Omron CX-Programmer project NuevoProyecto (CX-Programmer ?)

# PLC NuevoPLC1: CPM1(CPM1A) CPU30

## Program NuevoPrograma1 (no task)
Local symbols
TIM BOOL

### Section Sección1

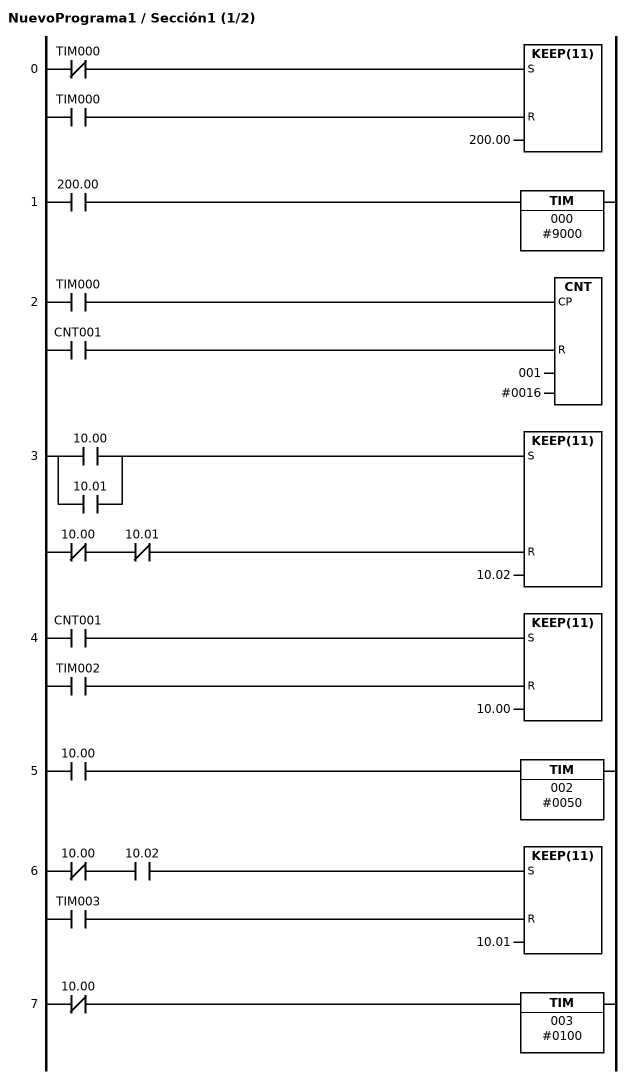
; rung 0
LDNOT TIM000
LD TIM000
KEEP(11) 200.00
; rung 1
LD 200.00
TIM 000 #9000  // Cuenta 15 minutos
; rung 2
LD TIM000
LD CNT001
CNT 001 #0016  // 15 min*16 iter = 4 Horas
; rung 3
LD 10.00
OR 10.01
LDNOT 10.00
ANDNOT 10.01
KEEP(11) 10.02  // KM3 (Motor comida)
; rung 4
LD CNT001
LD TIM002
KEEP(11) 10.00  // EV1 (Regula la entrada de comida al depósito)
; rung 5
LD 10.00
TIM 002 #0050  // Cuenta 5 seg
; rung 6
LDNOT 10.00
AND 10.02
LD TIM003
KEEP(11) 10.01  // EV2 (Regula la entrada de comida al agua)
; rung 7
LDNOT 10.00
TIM 003 #0100  // Cuenta 10 seg

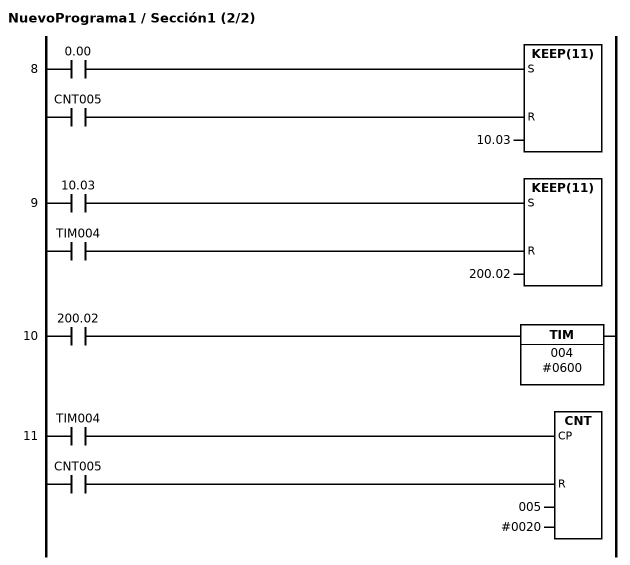
; rung 8
LD 0.00  // Sensor nivel de oxígeno (O2)
LD CNT005
KEEP(11) 10.03  // Bomba (Oxigena el agua)
; rung 9
LD 10.03
LD TIM004
KEEP(11) 200.02
; rung 10
LD 200.02
TIM 004 #0600  // Cuenta 60 seg
; rung 11
LD TIM004
LD CNT005
CNT 005 #0020  // 60 seg * 20 iter = 20 min
; rung 12
END(01)